FUNCTION_BLOCK AX_TO_AB (* Composite FB for converting AX (BOOL) adapter to AB (BYTE) adapter — bit-reinterpretation (structural copy between bit-string types; truncates on narrowing, zero-extends on widening). *)
  (* Standard: 61499-2; Description: Copyright (c) 2026 HR Agrartechnik GmbH This program and the accompanying materials are made available under the terms of the Eclipse Public License 2.0 which is available at https://www.eclipse.org/legal/epl-2.0/ SPDX-License-Identifier: EPL-2.0 *)
  (* Version 1.0, 2026-02-17, Franz Höpfinger, HR Agrartechnik GmbH *)
  PACKAGE adapter::conversion::unidirectional;
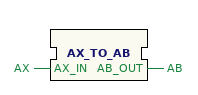
  SOCKETS
    AX_IN : adapter::types::unidirectional::AX; (* BOOL Adapter Input *)
  END_SOCKETS
  PLUGS
    AB_OUT : adapter::types::unidirectional::AB; (* BYTE Adapter Output *)
  END_PLUGS
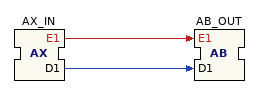
  EVENT_CONNECTIONS
    AX_IN.E1 TO AB_OUT.E1;
  END_CONNECTIONS
  DATA_CONNECTIONS
    AX_IN.D1 TO AB_OUT.D1;
  END_CONNECTIONS
END_FUNCTION_BLOCK
